(* CODESYS project IoDrvTemplateTest.project

Project tree, tasks and I/O mapping:
  CodesysControl : CoDeSys Control Win V3, 3S - Smart Software Solutions GmbH, version 3.5.0.0
    application Application
      task T1 (cyclic, interval t#20ms, priority 1) calls Main
      program POU_MyCard_1 [ST]
      program POU_MyCard_2 [ST]
      program Main [ST]
    MyCard_1 : MyCard, MyCompany, version 3.5.4.0
        input  dwIn0 : TChannel4Byte  // in1
        output bOut0_0 : BOOL  // out1.Byte0.Bit0
        output bOut0_1 : BOOL  // out1.Byte0.Bit1
        output bOut0_2 : BOOL  // out1.Byte0.Bit2
        output bOut0_3 : BOOL  // out1.Byte0.Bit3
        output bOut0_4 : BOOL  // out1.Byte0.Bit4
        output bOut0_5 : BOOL  // out1.Byte0.Bit5
        output bOut0_6 : BOOL  // out1.Byte0.Bit6
        output bOut0_7 : BOOL  // out1.Byte0.Bit7
        output bOut1_0 : BOOL  // out1.Byte1.Bit0
        output bOut1_1 : BOOL  // out1.Byte1.Bit1
        output bOut1_2 : BOOL  // out1.Byte1.Bit2
        output bOut1_3 : BOOL  // out1.Byte1.Bit3
        output bOut1_4 : BOOL  // out1.Byte1.Bit4
        output bOut1_5 : BOOL  // out1.Byte1.Bit5
        output bOut1_6 : BOOL  // out1.Byte1.Bit6
        output bOut1_7 : BOOL  // out1.Byte1.Bit7
        output bOut2_0 : BOOL  // out1.Byte2.Bit0
        output bOut2_1 : BOOL  // out1.Byte2.Bit1
        output bOut2_2 : BOOL  // out1.Byte2.Bit2
        output bOut2_3 : BOOL  // out1.Byte2.Bit3
        output bOut2_4 : BOOL  // out1.Byte2.Bit4
        output bOut2_5 : BOOL  // out1.Byte2.Bit5
        output bOut2_6 : BOOL  // out1.Byte2.Bit6
        output bOut2_7 : BOOL  // out1.Byte2.Bit7
        output bOut3_0 : BOOL  // out1.Byte3.Bit0
        output bOut3_1 : BOOL  // out1.Byte3.Bit1
        output bOut3_2 : BOOL  // out1.Byte3.Bit2
        output bOut3_3 : BOOL  // out1.Byte3.Bit3
        output bOut3_4 : BOOL  // out1.Byte3.Bit4
        output bOut3_5 : BOOL  // out1.Byte3.Bit5
        output bOut3_6 : BOOL  // out1.Byte3.Bit6
        output bOut3_7 : BOOL  // out1.Byte3.Bit7
        unmapped channels: out1
    MyCard_2 : MyCard, MyCompany, version 3.5.4.0
        input  dwIn10 : TChannel4Byte  // in1
        output bOut10_0 : BOOL  // out1.Byte0.Bit0
        output bOut10_1 : BOOL  // out1.Byte0.Bit1
        output bOut10_2 : BOOL  // out1.Byte0.Bit2
        output bOut10_3 : BOOL  // out1.Byte0.Bit3
        output bOut10_4 : BOOL  // out1.Byte0.Bit4
        output bOut10_5 : BOOL  // out1.Byte0.Bit5
        output bOut10_6 : BOOL  // out1.Byte0.Bit6
        output bOut10_7 : BOOL  // out1.Byte0.Bit7
        output bOut11_0 : BOOL  // out1.Byte1.Bit0
        output bOut11_1 : BOOL  // out1.Byte1.Bit1
        output bOut11_2 : BOOL  // out1.Byte1.Bit2
        output bOut11_3 : BOOL  // out1.Byte1.Bit3
        output bOut11_4 : BOOL  // out1.Byte1.Bit4
        output bOut11_5 : BOOL  // out1.Byte1.Bit5
        output bOut11_6 : BOOL  // out1.Byte1.Bit6
        output bOut11_7 : BOOL  // out1.Byte1.Bit7
        output bOut12_0 : BOOL  // out1.Byte2.Bit0
        output bOut12_1 : BOOL  // out1.Byte2.Bit1
        output bOut12_2 : BOOL  // out1.Byte2.Bit2
        output bOut12_3 : BOOL  // out1.Byte2.Bit3
        output bOut12_4 : BOOL  // out1.Byte2.Bit4
        output bOut12_5 : BOOL  // out1.Byte2.Bit5
        output bOut12_6 : BOOL  // out1.Byte2.Bit6
        output bOut12_7 : BOOL  // out1.Byte2.Bit7
        output bOut13_0 : BOOL  // out1.Byte3.Bit0
        output bOut13_1 : BOOL  // out1.Byte3.Bit1
        output bOut13_2 : BOOL  // out1.Byte3.Bit2
        output bOut13_3 : BOOL  // out1.Byte3.Bit3
        output bOut13_4 : BOOL  // out1.Byte3.Bit4
        output bOut13_5 : BOOL  // out1.Byte3.Bit5
        output bOut13_6 : BOOL  // out1.Byte3.Bit6
        output bOut13_7 : BOOL  // out1.Byte3.Bit7
        unmapped channels: out1
*)

// CodesysControl/Application/Main
PROGRAM Main
VAR
	A : DINT;
END_VAR

A := A + 1;

POU_MyCard_1();
POU_MyCard_2();

END_PROGRAM

// CodesysControl/Application/POU_MyCard_1
PROGRAM POU_MyCard_1
VAR
	In : ARRAY [0..3] OF BYTE;
	Out0 : BYTE := 2#01010101;
	Out1 : BYTE := 2#00110011;
	Out2 : BYTE := 2#00001111;
	Out3 : BYTE := 2#11110000;
END_VAR

In[0] := dwIn0.Byte0;
In[1] := dwIn0.Byte1;
In[2] := dwIn0.Byte2;
In[3] := dwIn0.Byte3;

bOut0_0 := Out0.0;
bOut0_1 := Out0.1;
bOut0_2 := Out0.2;
bOut0_3 := Out0.3;
bOut0_4 := Out0.4;
bOut0_5 := Out0.5;
bOut0_6 := Out0.6;
bOut0_7 := Out0.7;

bOut1_0 := Out1.0;
bOut1_1 := Out1.1;
bOut1_2 := Out1.2;
bOut1_3 := Out1.3;
bOut1_4 := Out1.4;
bOut1_5 := Out1.5;
bOut1_6 := Out1.6;
bOut1_7 := Out1.7;

bOut2_0 := Out2.0;
bOut2_1 := Out2.1;
bOut2_2 := Out2.2;
bOut2_3 := Out2.3;
bOut2_4 := Out2.4;
bOut2_5 := Out2.5;
bOut2_6 := Out2.6;
bOut2_7 := Out2.7;

bOut3_0 := Out3.0;
bOut3_1 := Out3.1;
bOut3_2 := Out3.2;
bOut3_3 := Out3.3;
bOut3_4 := Out3.4;
bOut3_5 := Out3.5;
bOut3_6 := Out3.6;
bOut3_7 := Out3.7;

END_PROGRAM

// CodesysControl/Application/POU_MyCard_2
PROGRAM POU_MyCard_2
VAR
	In : ARRAY [0..3] OF BYTE;
	Out10 : BYTE := 2#11110000;
	Out11 : BYTE := 2#00110011;
	Out12 : BYTE := 2#00001111;
	Out13 : BYTE := 2#01010101;
END_VAR

In[0] := dwIn10.Byte0;
In[1] := dwIn10.Byte1;
In[2] := dwIn10.Byte2;
In[3] := dwIn10.Byte3;

bOut10_0 := Out10.0;
bOut10_1 := Out10.1;
bOut10_2 := Out10.2;
bOut10_3 := Out10.3;
bOut10_4 := Out10.4;
bOut10_5 := Out10.5;
bOut10_6 := Out10.6;
bOut10_7 := Out10.7;

bOut11_0 := Out11.0;
bOut11_1 := Out11.1;
bOut11_2 := Out11.2;
bOut11_3 := Out11.3;
bOut11_4 := Out11.4;
bOut11_5 := Out11.5;
bOut11_6 := Out11.6;
bOut11_7 := Out11.7;

bOut12_0 := Out12.0;
bOut12_1 := Out12.1;
bOut12_2 := Out12.2;
bOut12_3 := Out12.3;
bOut12_4 := Out12.4;
bOut12_5 := Out12.5;
bOut12_6 := Out12.6;
bOut12_7 := Out12.7;

bOut13_0 := Out13.0;
bOut13_1 := Out13.1;
bOut13_2 := Out13.2;
bOut13_3 := Out13.3;
bOut13_4 := Out13.4;
bOut13_5 := Out13.5;
bOut13_6 := Out13.6;
bOut13_7 := Out13.7;

END_PROGRAM
